TYPE ST_ERROR_LOG :
STRUCT
	sTimeOfError:					STRING;
	eErrorCode:						E_CIM_ERROR_CODES;
//	bErrorCleared:					BOOL;
END_STRUCT
END_TYPE

(* stored: Version 1.1.0.1, ProductVersion 3.1.4024.12
   DUT ST_ERROR_LOG: Id {3edb04cf-c447-4fa8-90ea-190cb0003c98} *)
